FUNCTION_BLOCK NewBatch EXTENDS BaseState
VAR_INPUT
END_VAR
VAR_OUTPUT
END_VAR
VAR
END_VAR

METHOD mIrun : BOOL
IF BasePointer^.MachineFlagsAccessI.pBuffering = TRUE THEN
	BasePointer^.MachineFlagsAccessI.pHaltBatch := TRUE;
ELSE
	BasePointer^.MachineFlagsAccessI.pHaltBatch := FALSE;
	mNextState();	
END_IF
END_METHOD

END_FUNCTION_BLOCK

(* stored: Version 1.1.0.1, ProductVersion 3.1.4024.12
   POU NewBatch: Id {5cf4f6aa-ca64-4d77-a407-cbbaafb258d5}, SpecialFunc None
   Method mIrun: Id {dc1f69bf-216a-4a80-a7cb-a8fb864039d2} *)
